Universal Robots PolyScope program: Robot 3 12_10.urp

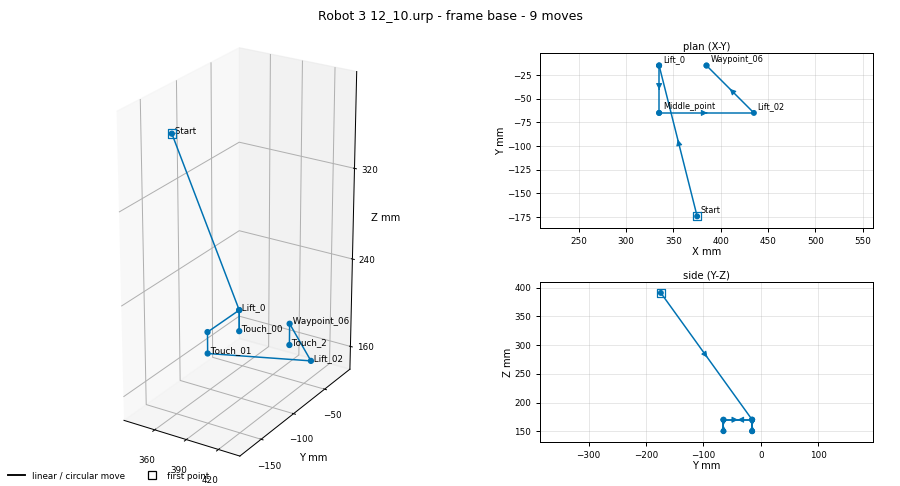
[picture p0: tool path of Robot 3 12_10.urp in frame base, 9 of 9 moves have a stored position in this frame; points joined in program order, loops and branches not executed]
Program Robot 3 12_10 (installation=default directory=/programs createdIn=5.12.2.1101534 lastSavedIn=5.11.9.1010452 robotSerialNumber=20225200364)
Calibrated DH parameters: a=[0.00002, -0.569483, -0.54992, -0.00001, -0.000036, 0]; d=[0.180894, -146.691669, 192.918669, -46.053088, 0.119778, 0.115602]; alpha=[1.571425, -0.001534, 0.003359, 1.568739, -1.571477, 0]; deltaTheta=[0, 0.376258, -0.101074, -0.275185, -0.000002, 0]
Robot Program (runOnlyOnce=false)
  MoveL speed 250 mm/s, acceleration 1200 mm/s^2 (useActiveTCP=true) feature=Base
    Waypoint Start: TCP in base x=375.127 y=-174.15 z=391.075 mm, rx=2.2214 ry=2.2214 rz=0 rad; joints [0, -90, -120, -240, -90, 0] deg
    Waypoint Lift_0: TCP in base x=334.998 y=-15 z=170 mm, rx=2.2214 ry=2.2214 rz=0 rad; joints [28.724, -101.341, -138.641, -210.018, -90, 28.724] deg
    Waypoint Touch_00: motionParameters(jointSpeed=1.047198 jointAcceleration=1.396263 cartesianSpeed=0.005 cartesianAcceleration=1.2); TCP in base x=335 y=-15 z=150 mm, rx=2.2214 ry=2.2214 rz=0 rad; joints [28.724, -103.84, -139.118, -207.042, -90, 28.724] deg
      Until TOOL_CONTACT_DETECTION (allowActions=false retraction=-0.0003 decelerationAcceleration=3 decelerationAngularAcceleration=34.906585)
    MoveDirectionNode (selectedDirection=YMinus)
      Until DISTANCE (allowActions=false deceleration=3 distanceNodeType=STOP) Distance=0.1; motionParameters(blendRadius=0)
    MoveDirectionNode (selectedDirection=XPlus)
      Until DISTANCE (allowActions=false deceleration=3 distanceNodeType=STOP) Distance=0.1; motionParameters(blendRadius=0)
    MoveDirectionNode (selectedDirection=YPlus)
      Until DISTANCE (allowActions=false deceleration=3 distanceNodeType=STOP) Distance=0.1; motionParameters(blendRadius=0)
    MoveDirectionNode (selectedDirection=XMinus)
      Until DISTANCE (allowActions=false deceleration=3 distanceNodeType=STOP) Distance=0.1; motionParameters(blendRadius=0)
    Waypoint Lift_01: TCP in base x=334.998 y=-15 z=170 mm, rx=2.2214 ry=2.2214 rz=0 rad; joints [28.724, -101.341, -138.641, -210.018, -90, 28.724] deg
    Waypoint Middle_point: TCP in base x=334.998 y=-65 z=170 mm, rx=2.2214 ry=2.2214 rz=0 rad; joints [19.706, -101.827, -137.946, -210.227, -90, 19.706] deg
    Waypoint Touch_01: TCP in base x=334.998 y=-65 z=150 mm, rx=2.2214 ry=2.2214 rz=0 rad; joints [19.706, -104.286, -138.416, -207.297, -90, 19.706] deg
    MoveDirectionNode (selectedDirection=XPlus)
      Until DISTANCE (allowActions=false deceleration=3 distanceNodeType=STOP) Distance=0.1; motionParameters(blendRadius=0)
    Waypoint Lift_02: TCP in base x=434.998 y=-65 z=170 mm, rx=2.2214 ry=2.2214 rz=0 rad; joints [14.827, -109.269, -126.497, -214.234, -90, 14.827] deg
    Waypoint Waypoint_06: TCP in base x=384.998 y=-15 z=170 mm, rx=2.2214 ry=2.2214 rz=0 rad; joints [24.641, -105.278, -132.815, -211.907, -90, 24.641] deg
    Waypoint Touch_2: TCP in base x=384.998 y=-15 z=150 mm, rx=2.2214 ry=2.2214 rz=0 rad; joints [24.641, -107.481, -133.244, -209.275, -90, 24.641] deg
    MoveDirectionNode (selectedDirection=YMinus)
      Until DISTANCE (allowActions=false deceleration=3 distanceNodeType=STOP) Distance=0.1; motionParameters(blendRadius=0)
